PROGRAM ReceiveSwitch
VAR
	fbReceiveSwitchMessage: FB_Rec_RPS_Switch;
END_VAR

fbReceiveSwitchMessage(
	str_KL6581:= EnOcean.stBuffer, 
	byNode:= 0, 
	dw_ID:= EnOcean.dwSwitchID, 
	str_EnOceanSwitch=> EnOcean.stSwitchData, 
	by_Node=> , 
	bReceive=> EnOcean.bSwitchDataReceived);

END_PROGRAM

(* stored: Version 1.1.0.1, ProductVersion 3.1.4024.11
   POU ReceiveSwitch: Id {4437d9f6-ff2a-4f6c-8be8-1a136922cd63}, SpecialFunc None *)
